FUNCTION_BLOCK FB_Klep IMPLEMENTS ITF_Klep
VAR
    _cmdOpen : BOOL;   // laatst aangevraagde command
    _status  : BOOL;   // huidige status van de klep
	
	_UnitStatus : E_UnitStatus := E_UnitStatus.Ok;

	_prevCmdOpen : BOOL;
	tonPositionTimeout : TON;
END_VAR

//ik wou nog een bericht zetten in de git dus vandaar deze comment maar het ging erover dat ik problemen had met mergen en dat mijn alarmen die ik had gelust niet meer bestaan :) dus die ga ik morgen opnieuw bouwen maar daar heb ik nu geen zin in want het is bijna 2 uur s'avonds :) en waarom lees je dit hele bericht trouwens dat was echt een verspilling van je tijd :0 xoxo groetjes niek

METHOD ResetFault : BOOL
_UnitStatus := E_UnitStatus.Ok;
tonPositionTimeout(IN := FALSE);

ResetFault := TRUE;
END_METHOD

PROPERTY PUBLIC Status : BOOL
GET
Status := _status;   // status uitlezen
END_GET
SET
_status := Status;
END_SET
END_PROPERTY

METHOD PUBLIC SturingOpen : BOOL
VAR_INPUT
	i_bOpen	: BOOL; // TRUE = open, FALSE = dicht
END_VAR
_cmdOpen := i_bOpen;

// als commando verandert: start timer om te checken of status volgt
IF _cmdOpen <> _prevCmdOpen THEN
	tonPositionTimeout(IN := TRUE, PT := T#2S);
END_IF

// als status overeenkomt met commando: klaar -> timer uit, status OK (maar alleen als nog geen error latched is)
IF _status = _cmdOpen THEN
	tonPositionTimeout(IN := FALSE);
	IF _UnitStatus <> E_UnitStatus.Error THEN
		_UnitStatus := E_UnitStatus.Ok;
	END_IF
END_IF

// als timer afloopt en status volgt nog niet: error latched
IF tonPositionTimeout.Q THEN
	_UnitStatus := E_UnitStatus.Error;
	tonPositionTimeout(IN := FALSE);
END_IF

_prevCmdOpen := _cmdOpen;

SturingOpen := TRUE;
END_METHOD

PROPERTY UnitStatus : E_UnitStatus
GET
UnitStatus := _UnitStatus;
END_GET
SET
_UnitStatus := UnitStatus;
END_SET
END_PROPERTY

END_FUNCTION_BLOCK

(* stored: Version 1.1.0.1
   POU FB_Klep: Id {a42b2b1d-3d0d-4ad8-8a49-e659df0386f5}, SpecialFunc None
   Folder Methods: Id {215c97dc-4785-4f3f-80d3-672f5b9c53d7}
   Folder Properties: Id {8948e215-6589-49b0-8016-a5dec4d22119}
   Method ResetFault: Id {4d351831-0df5-4419-82cc-7a21b8bbdd9c}
   Property Status: Id {fac60b85-9052-4a73-9fa5-0cc4b71f46f0}
   Get Get: Id {126ac777-00b4-45e9-900d-48260272a880}
   Set Set: Id {52aaba85-13ed-4e62-a0db-c488bafb88d7}
   Method SturingOpen: Id {789bb220-7b95-473c-9a9f-a5eb352b7b20}
   Property UnitStatus: Id {ea2a5305-b813-4fa3-8406-0429b7a3d583}
   Get Get: Id {16bdf221-79b6-451b-9242-4cf56e2054de}
   Set Set: Id {8401844a-397f-46ac-961b-ea0dc10d9123} *)
